FUNCTION_BLOCK FB_MotionRef
VAR_INPUT
	fTime : LREAL;
	fAmplitude : LREAL;
	fFrequency : LREAL;
	fInitialPos : LREAL;
END_VAR
VAR_OUTPUT
	fXDotRef : LREAL;
	fXRef : LREAL;
END_VAR
VAR
	fPI : LREAL := 3.1415;
	fMean : LREAL;
END_VAR

fMean := fAmplitude + fInitialPos; 
IF G_Inputs.bStartButton THEN
	fXRef := fMean - fAmplitude * COS(2*fPI * fFrequency * fTime);
	fXDotRef := 2 * fPI *fFrequency * fAmplitude * SIN(2*fPI * fFrequency * fTime);
ELSE
	fXDotRef := 0.0;
END_IF

END_FUNCTION_BLOCK

(* stored: Version 1.1.0.1, ProductVersion 3.1.4024.12
   POU FB_MotionRef: Id {354b3a34-d392-4f87-a4eb-f033618b096f}, SpecialFunc None *)
